(* CoDeSys 2.3.9.37 project: Cap8_3.pro *)
(* Libraries: Standard.lib 4.10.05 12:14:46 *)

(* Global variable list: Global_Variables *)
VAR_GLOBAL
     (* Entrada *)
     Habilita:BOOL;
     (* Salida *)
     Verde:BOOL;
     Ambar:BOOL;
      Rojo:BOOL;
END_VAR

(* POU PLC_PRG, LD *)
PROGRAM PLC_PRG
VAR

END_VAR
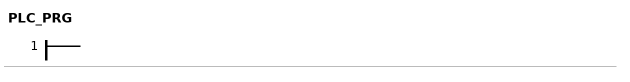
_LD_ (* Ladder Diagram *)
NETWORK 1
	*
_END_LD_
(* the same logic as Structured Text *)
(* Network 1 *)
END_PROGRAM

(* Visualisation Visu
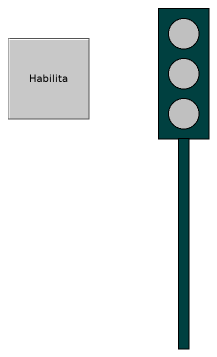
button at (20,50)-(101,131): text "Habilita"; toggles Habilita
ellipse at (180,30)-(211,61): alarm colour if Rojo
ellipse at (180,70)-(211,101): alarm colour if Ambar
ellipse at (180,110)-(211,141): alarm colour if Verde
2 more shapes without text or variables
*)
